FUNCTION_BLOCK M_SOLVE (* Solve the matrix equation IN1*OUT=IN2 for OUT *)
  (* Standard: 61499-1; Classification: Matrix Operations; Function: Inversion *)
  (* Version 0.0, 2008-07-07, JHC, Holobloc Inc, Changed to single IN1 input. *)
  (* Compiler header: package fb.rt.math.matrix; *)
  (* Compiler classdef: public class M_MUL extends M_ADD *)
  (* Compiler Java Sun JDK 1.6.0 *)
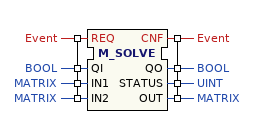
  EVENT_INPUT
    REQ WITH QI, IN1, IN2; (* Solve IN1*OUT=IN2 for OUT *)
  END_EVENT
  EVENT_OUTPUT
    CNF WITH QO, STATUS, OUT; (* Confirmation of Requested Service *)
  END_EVENT
  VAR_INPUT
    QI : BOOL; (* Event Input Qualifier *)
    IN1 : MATRIX; (* Matrix to be inverted - unaffected by inversion operation *)
    IN2 : MATRIX;
  END_VAR
  VAR_OUTPUT
    QO : BOOL; (* Event Output Qualifier *)
    STATUS : UINT; (* 0=OK, 4=DIVISION_BY_0, 13=ARRAY_SIZE_ERROR *)
    OUT : MATRIX; (* Inverse of IN1 *)
  END_VAR
END_FUNCTION_BLOCK
